Staubli VAL3: onF7Event.pgx

program onF7Event()
  local num l_nResult
  local bool l_bYes
  local string l_sMessage
  local string l_sMessage2
  local string l_sButton[2]
  local string l_sName
  local string l_sAction
  local num l_nSize
  local num i
  local num l_nSizeAction
  local num j
  local string l_sItem
  local InstrItem l_iItem
  local string l_sProgSwap
  local bool l_bFound
begin
  // look if the bButton is enable
  if bButton[6]
    //
    // DELETE
    //
    // do not delete HOME1 HOME2
    if sEvent=="HOME1" or sEvent=="HOME2"
      call language:message(l_sMessage,23)
      popUpMsg(l_sMessage+" "+sEvent)
    elseIf sEvent!=""
      // look inside the process List
      call processList:isFound(sEvent,l_bFound)
      if !l_bFound
        // scan inside all the program
        l_sName=sEvent
        l_iItem.sType=l_sProgSwap=sProgType
        l_iItem.sData=sEvent
        if l_sProgSwap!="PROG"
          // reload the program as default
          sProgType="PROG"
          // load the progType
          call load()
        endIf
        // find it
        call prog:findItem(l_iItem,l_nResult,false)
        if l_sProgSwap!="PROG"
          // reload the program as default
          sProgType=l_sProgSwap
          // load the progType
          call load()
        endIf
      endIf
      // if not found
      if l_nResult==0 and !l_bFound
        call language:message(l_sMessage,22)
        // get the yes_no button Key
        call language:getYesNo(l_sButton)
        // ask the question
        call use:yes_no(l_sMessage+sEvent,l_sButton,l_bYes)
        if l_bYes
          call prog:delete(sEvent,l_nResult)
          if l_nResult==0
            logMsg("[KERNEL] INTERFACE:Delete the program: "+sEvent)
            call buildList()
          else
            popUpMsg("error code: "+toString("",l_nResult))
            logMsg("[KERNEL] INTERFACE:Delete the program: "+sEvent+"error code: "+toString("",l_nResult))
          endIf
        endIf
      elseIf l_bFound
        // the program is in the processList
        call language:message(l_sMessage,23)
        call language:message(l_sMessage2,24)
        popUpMsg(l_sMessage+l_sMessage2)
      endIf
    endIf
  endIf
end
